FUNCTION_BLOCK FB_BinaryInp
VAR_INPUT
	bPush : BOOL;
	bReset : BOOL;
END_VAR
VAR_OUTPUT
	bOutActive : BOOL;
END_VAR
VAR
	rsHold : RS;
END_VAR

rsHold(SET:=bPush, RESET1:=bReset, Q1=>bOutActive);

END_FUNCTION_BLOCK

(* stored: Version 1.1.0.1, ProductVersion 3.1.4024.6
   POU FB_BinaryInp: Id {7c991cde-f35e-49c7-832a-d3659d6f05da}, SpecialFunc None *)
